# EPICS autosave request: kinetixApp/Db/ADKinetix_settings.req
file "ADBase_settings.req", P=$(P), R=$(R)
$(P)$(R)UniqueIdMode
